(* CODESYS project wago_ecternal_python_script_example_v0.0.1.ecp

Project tree, tasks and I/O mapping:
  PFC200_2ETH_CAN : 750-8203 PFC200 2ETH CAN, WAGO, order no. 0750-8203, version 5.11.1.16
    application Application
      libraries: ; SysProcess, 3.5.7.0 (System); ISysTypes2, 3.5.0.0 (System); WagoLibPythonExternalFile, 0.0.1 (WAGO Corp. USA)
      task PLC_Task (cyclic, interval t#50ms, priority 15) calls PLC_PRG
      program PLC_PRG [ST]
      EcPyTest
    DeviceAdapter
    Kbus : Kbus, WAGO, version 1.4.0.2
        unmapped channels: K-BUS diagnostics
      _16_DO_Generic : 075x-16DO, WAGO, order no. 075x-16DO, version 0.0.0.13
          settings: K-BUS Module slot index = 1
          unmapped channels: _OUT
        DeviceAdapter
    MODBUS
      MODBUS : MODBUS, WAGO, order no. n/a, version 1.1.1.15
    CANbus
  00000000-0000-0000-0000-000000000000|Z:\Dropbox\Demos\e!Cockpit\Python\Python Script\EcPyTest.py
*)

// PFC200_2ETH_CAN/Application/PLC_PRG
PROGRAM PLC_PRG
VAR	
	fbPy				: WagoLibPythonExternalFile.fbPythonCall;
	xPyGo				: BOOL;
	asPyArgv			: ARRAY[0..1] OF STRING := ['123', '456'];
	sFileName			: STRING := 'EcPyTest.py';
	sPyRtn				: STRING;
END_VAR

//toggle the xPyGo BOOL to execute the python script
fbPy(xExecute:= xPyGo, 
	asArgv:= asPyArgv, 
	sFileName:= sFileName, 
	sReturnData=> sPyRtn);

END_PROGRAM
